Fanuc KAREL source: BYNAME.kl

PROGRAM T
%NOLOCKGROUP
VAR
 v0 : STRING[40]
 v1 : STRING[40]
 v2 : INTEGER
BEGIN
 BYNAME(v0, v1, v2)
END T
